// TIA Portal V16 export
// export: Created 2021-11-12T13:31:47.3064744Z, ExportSetting WithDefaults, DisplayName Totally Integrated Automation Portal, DisplayVersion V16 Update 3, DisplayName TIA Portal Version Control Interface, DisplayVersion V16 Update 2, DisplayName TIA Portal Openness, DisplayVersion V16 Update 3, DisplayName SINAMICS Startdrive Advanced, DisplayVersion V16 Update 5, DisplayName SINAMICS Startdrive G130, G150, S120, S150, SINAMICS MV, S210, DisplayVersion V16 Update 5, DisplayName SINAMICS Startdrive G110M, G120, G120C, G120D, G120P, G115D, DisplayVersion V16 Update 5, DisplayName STEP 7 Professional, DisplayVersion V16 Update 3, DisplayName STEP 7 Safety, DisplayVersion V16, DisplayName WinCC UA Professional, DisplayVersion V16 Update 3
FUNCTION_BLOCK "Zone000"   // FB72, LAD
{ S7_Optimized_Access := 'TRUE' }
VERSION : 0.1
// stored: AutoNumber true, IsIECCheckEnabled false, IsRetainMemResEnabled false, MemoryReserve 100, SetENOAutomatically false, UDAEnableTagReadback false
   VAR
      SF_StationMEM1Mode { S7_SetPoint := 'True'} : "STD_Station";
      "SF_EQ01-MA01" : "STD_Drive1";   // Čerpadlo cirkulace (P133) / Water pump (P51)
      "SF_EQ01-MA02" : "STD_Drive1";   // Čerpadlo cirkulace (P133) / Water pump (P52)
      "SF_EQ02-MA01" : "STD_Drive1";   // Čerpadlo cirkulace (P133) / Water pump (P61)
      "SF_UC11-TA01" { S7_SetPoint := 'True'} : "STD_Siemens_G120_CU240E_2_PN";   // Frekvenční měnič ( pro P33) / Frequence changer
      "SF_UC11-TA02" { S7_SetPoint := 'True'} : "STD_Siemens_G120_CU240E_2_PN";   // Frekvenční měnič ( pro P33) / Frequence changer
      "SF_UC11-TA03" { S7_SetPoint := 'True'} : "STD_Siemens_G120_CU240E_2_PN";   // Frekvenční měnič ( pro P33) / Frequence changer
      SS_Edge { S7_SetPoint := 'True'} : Array[0..100] of Bool;
      SB1_PowerOk { S7_SetPoint := 'True'} : Bool;
   END_VAR
   VAR_TEMP
      TS_EQ01MA01 : "UDT_DriveControl";   // Water pump (P51) / Čerpadlo cirkulace (P133)
      TS_EQ01MA02 : "UDT_DriveControl";   // Valve with servomotor (P52) / Ventil se servopohonem (A1419)
      TS_EQ02MA01 : "UDT_DriveControl";   // Valve with servomotor (P61) / Ventil se servopohonem (A1416)
      TS_UC11TA01 : Struct   // Frequence changer / Frekvenční měnič ( pro P33)
         ReqDir1 : Bool;   // Move in direction 1
         ReqDir2 : Bool;   // Move in direction 2
         AckErr : Bool;   // Acknowledge error
         SpeedSP : Real;   // Speed setpoint
      END_STRUCT;
      TS_UC11TA02 : Struct   // Frequence changer / Frekvenční měnič ( pro P33)
         ReqDir1 : Bool;   // Move in direction 1
         ReqDir2 : Bool;   // Move in direction 2
         AckErr : Bool;   // Acknowledge error
         SpeedSP : Real;   // Speed setpoint
      END_STRUCT;
      TS_UC11TA03 : Struct   // Frequence changer / Frekvenční měnič ( pro P33)
         ReqDir1 : Bool;   // Move in direction 1
         ReqDir2 : Bool;   // Move in direction 2
         AckErr : Bool;   // Acknowledge error
         SpeedSP : Real;   // Speed setpoint
      END_STRUCT;
   END_VAR
BEGIN

REGION Network 1: *************** Zone 000 ***************
END_REGION

REGION Network 2: Acknowledge from all zones
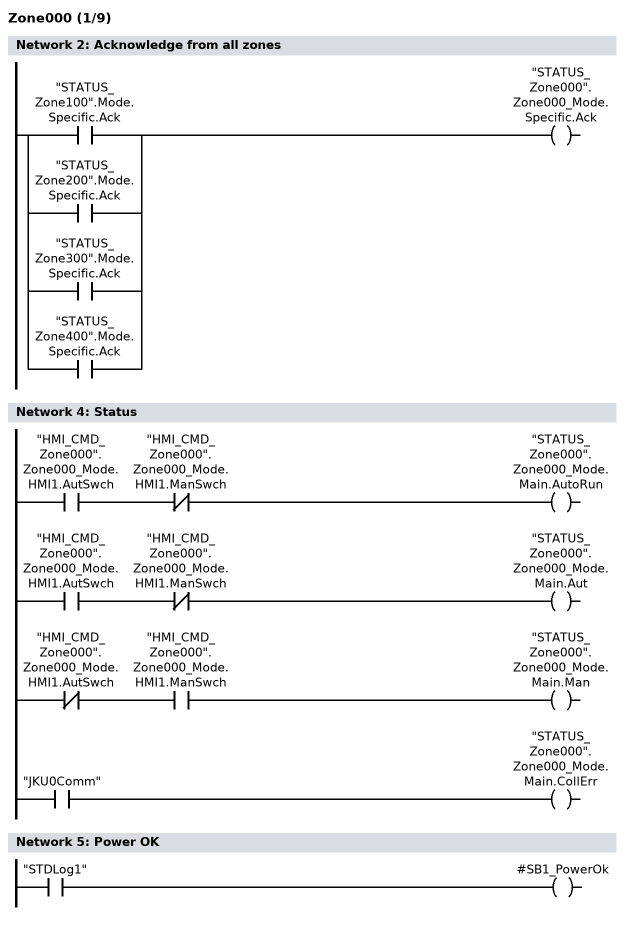
   RUNG wire#powerrail
      Contact( "STATUS_Zone100".Mode.Specific.Ack )
      wire#w1
      Coil( "STATUS_Zone000".Zone000_Mode.Specific.Ack )
   END_RUNG
   RUNG wire#powerrail
      Contact( "STATUS_Zone200".Mode.Specific.Ack )
   END_RUNG wire#w1
   RUNG wire#powerrail
      Contact( "STATUS_Zone300".Mode.Specific.Ack )
   END_RUNG wire#w1
   RUNG wire#powerrail
      Contact( "STATUS_Zone400".Mode.Specific.Ack )
   END_RUNG wire#w1
   // the same network as SCL:
   "STATUS_Zone000".Zone000_Mode.Specific.Ack := "STATUS_Zone100".Mode.Specific.Ack OR "STATUS_Zone200".Mode.Specific.Ack OR "STATUS_Zone300".Mode.Specific.Ack OR "STATUS_Zone400".Mode.Specific.Ack;
END_REGION

REGION Network 3: Alarms
END_REGION

REGION Network 4: Status
   RUNG wire#powerrail
      Contact( "HMI_CMD_Zone000".Zone000_Mode.HMI1.AutSwch )
      I_Contact( "HMI_CMD_Zone000".Zone000_Mode.HMI1.ManSwch )
      Coil( "STATUS_Zone000".Zone000_Mode.Main.AutoRun )
   END_RUNG
   RUNG wire#powerrail
      Contact( "HMI_CMD_Zone000".Zone000_Mode.HMI1.AutSwch )
      I_Contact( "HMI_CMD_Zone000".Zone000_Mode.HMI1.ManSwch )
      Coil( "STATUS_Zone000".Zone000_Mode.Main.Aut )
   END_RUNG
   RUNG wire#powerrail
      I_Contact( "HMI_CMD_Zone000".Zone000_Mode.HMI1.AutSwch )
      Contact( "HMI_CMD_Zone000".Zone000_Mode.HMI1.ManSwch )
      Coil( "STATUS_Zone000".Zone000_Mode.Main.Man )
   END_RUNG
   RUNG wire#powerrail
      Contact( "JKU0Comm" )
      Coil( "STATUS_Zone000".Zone000_Mode.Main.CollErr )
   END_RUNG
   // the same network as SCL:
   "STATUS_Zone000".Zone000_Mode.Main.AutoRun := "HMI_CMD_Zone000".Zone000_Mode.HMI1.AutSwch AND NOT "HMI_CMD_Zone000".Zone000_Mode.HMI1.ManSwch;
   "STATUS_Zone000".Zone000_Mode.Main.Aut := "HMI_CMD_Zone000".Zone000_Mode.HMI1.AutSwch AND NOT "HMI_CMD_Zone000".Zone000_Mode.HMI1.ManSwch;
   "STATUS_Zone000".Zone000_Mode.Main.Man := NOT "HMI_CMD_Zone000".Zone000_Mode.HMI1.AutSwch AND "HMI_CMD_Zone000".Zone000_Mode.HMI1.ManSwch;
   "STATUS_Zone000".Zone000_Mode.Main.CollErr := "JKU0Comm";
END_REGION

REGION Network 5: Power OK
   RUNG wire#powerrail
      Contact( "STDLog1" )
      Coil( #SB1_PowerOk )
   END_RUNG
   // the same network as SCL:
   #SB1_PowerOk := "STDLog1";
END_REGION

REGION Network 6: *************** MEM1 ***************
END_REGION

REGION Network 7: MEM1 - Main control
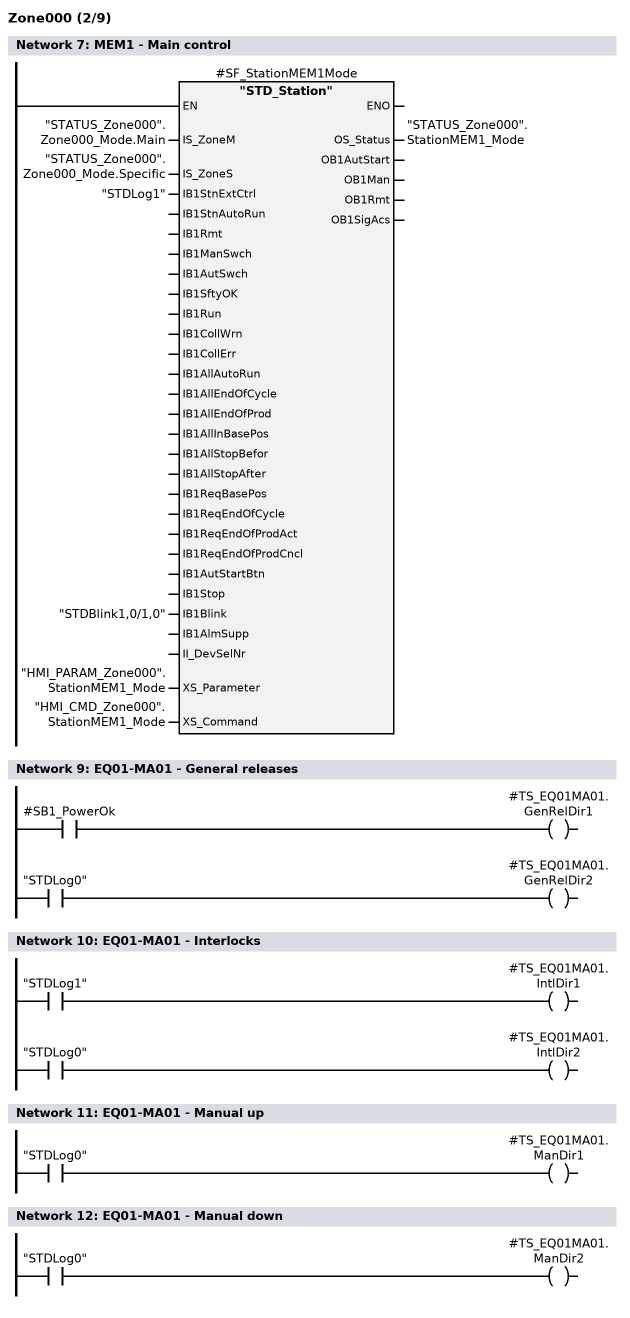
   RUNG wire#powerrail
      #SF_StationMEM1Mode(IS_ZoneM := "STATUS_Zone000".Zone000_Mode.Main, IS_ZoneS := "STATUS_Zone000".Zone000_Mode.Specific, IB1StnExtCtrl := "STDLog1", IB1StnAutoRun :=, IB1Rmt :=, IB1ManSwch :=, IB1AutSwch :=, IB1SftyOK :=, IB1Run :=, IB1CollWrn :=, IB1CollErr :=, IB1AllAutoRun :=, IB1AllEndOfCycle :=, IB1AllEndOfProd :=, IB1AllInBasePos :=, IB1AllStopBefor :=, IB1AllStopAfter :=, IB1ReqBasePos :=, IB1ReqEndOfCycle :=, IB1ReqEndOfProdAct :=, IB1ReqEndOfProdCncl :=, IB1AutStartBtn :=, IB1Stop :=, IB1Blink := "STDBlink1,0/1,0", IB1AlmSupp :=, II_DevSelNr :=, XS_Parameter := "HMI_PARAM_Zone000".StationMEM1_Mode, XS_Command := "HMI_CMD_Zone000".StationMEM1_Mode, OS_Status => "STATUS_Zone000".StationMEM1_Mode, OB1AutStart =>, OB1Man =>, OB1Rmt =>, OB1SigAcs =>)
   END_RUNG
   // the same network as SCL:
   #SF_StationMEM1Mode(IS_ZoneM := "STATUS_Zone000".Zone000_Mode.Main,   // "STD_Station"
                       IS_ZoneS := "STATUS_Zone000".Zone000_Mode.Specific,
                       IB1StnExtCtrl := "STDLog1",
                       IB1Blink := "STDBlink1,0/1,0",
                       XS_Parameter := "HMI_PARAM_Zone000".StationMEM1_Mode,
                       XS_Command := "HMI_CMD_Zone000".StationMEM1_Mode,
                       OS_Status => "STATUS_Zone000".StationMEM1_Mode);
END_REGION

REGION Network 8: ********** EQ01-MA01 **********
END_REGION

REGION Network 9: EQ01-MA01 - General releases
   RUNG wire#powerrail
      Contact( #SB1_PowerOk )
      Coil( #TS_EQ01MA01.GenRelDir1 )
   END_RUNG
   RUNG wire#powerrail
      Contact( "STDLog0" )
      Coil( #TS_EQ01MA01.GenRelDir2 )
   END_RUNG
   // the same network as SCL:
   #TS_EQ01MA01.GenRelDir1 := #SB1_PowerOk;
   #TS_EQ01MA01.GenRelDir2 := "STDLog0";
END_REGION

REGION Network 10: EQ01-MA01 - Interlocks
   RUNG wire#powerrail
      Contact( "STDLog1" )
      Coil( #TS_EQ01MA01.IntlDir1 )
   END_RUNG
   RUNG wire#powerrail
      Contact( "STDLog0" )
      Coil( #TS_EQ01MA01.IntlDir2 )
   END_RUNG
   // the same network as SCL:
   #TS_EQ01MA01.IntlDir1 := "STDLog1";
   #TS_EQ01MA01.IntlDir2 := "STDLog0";
END_REGION

REGION Network 11: EQ01-MA01 - Manual up
   RUNG wire#powerrail
      Contact( "STDLog0" )
      Coil( #TS_EQ01MA01.ManDir1 )
   END_RUNG
   // the same network as SCL:
   #TS_EQ01MA01.ManDir1 := "STDLog0";
END_REGION

REGION Network 12: EQ01-MA01 - Manual down
   RUNG wire#powerrail
      Contact( "STDLog0" )
      Coil( #TS_EQ01MA01.ManDir2 )
   END_RUNG
   // the same network as SCL:
   #TS_EQ01MA01.ManDir2 := "STDLog0";
END_REGION

REGION Network 13: EQ01-MA01 - Auto up
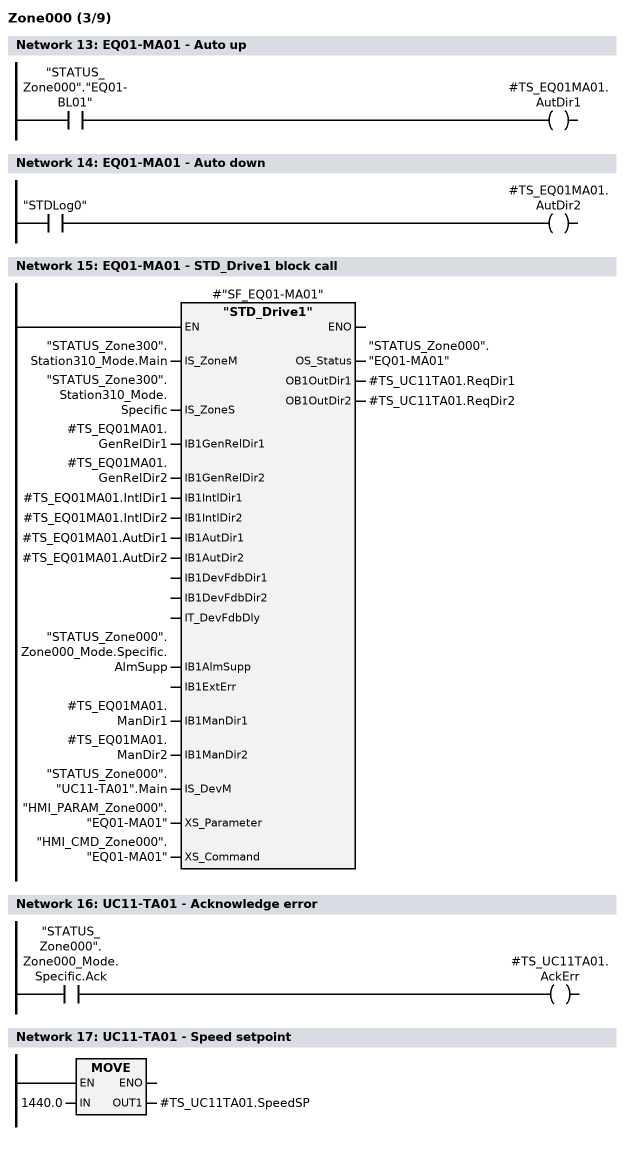
   RUNG wire#powerrail
      Contact( "STATUS_Zone000"."EQ01-BL01" )
      Coil( #TS_EQ01MA01.AutDir1 )
   END_RUNG
   // the same network as SCL:
   #TS_EQ01MA01.AutDir1 := "STATUS_Zone000"."EQ01-BL01";
END_REGION

REGION Network 14: EQ01-MA01 - Auto down
   RUNG wire#powerrail
      Contact( "STDLog0" )
      Coil( #TS_EQ01MA01.AutDir2 )
   END_RUNG
   // the same network as SCL:
   #TS_EQ01MA01.AutDir2 := "STDLog0";
END_REGION

REGION Network 15: EQ01-MA01 - STD_Drive1 block call
   RUNG wire#powerrail
      #"SF_EQ01-MA01"(IS_ZoneM := "STATUS_Zone300".Station310_Mode.Main, IS_ZoneS := "STATUS_Zone300".Station310_Mode.Specific, IB1GenRelDir1 := #TS_EQ01MA01.GenRelDir1, IB1GenRelDir2 := #TS_EQ01MA01.GenRelDir2, IB1IntlDir1 := #TS_EQ01MA01.IntlDir1, IB1IntlDir2 := #TS_EQ01MA01.IntlDir2, IB1AutDir1 := #TS_EQ01MA01.AutDir1, IB1AutDir2 := #TS_EQ01MA01.AutDir2, IB1DevFdbDir1 :=, IB1DevFdbDir2 :=, IT_DevFdbDly :=, IB1AlmSupp := "STATUS_Zone000".Zone000_Mode.Specific.AlmSupp, IB1ExtErr :=, IB1ManDir1 := #TS_EQ01MA01.ManDir1, IB1ManDir2 := #TS_EQ01MA01.ManDir2, IS_DevM := "STATUS_Zone000"."UC11-TA01".Main, XS_Parameter := "HMI_PARAM_Zone000"."EQ01-MA01", XS_Command := "HMI_CMD_Zone000"."EQ01-MA01", OS_Status => "STATUS_Zone000"."EQ01-MA01", OB1OutDir1 => #TS_UC11TA01.ReqDir1, OB1OutDir2 => #TS_UC11TA01.ReqDir2)
   END_RUNG
   // the same network as SCL:
   #"SF_EQ01-MA01"(IS_ZoneM := "STATUS_Zone300".Station310_Mode.Main,   // "STD_Drive1"
                   IS_ZoneS := "STATUS_Zone300".Station310_Mode.Specific,
                   IB1GenRelDir1 := #TS_EQ01MA01.GenRelDir1,
                   IB1GenRelDir2 := #TS_EQ01MA01.GenRelDir2,
                   IB1IntlDir1 := #TS_EQ01MA01.IntlDir1,
                   IB1IntlDir2 := #TS_EQ01MA01.IntlDir2,
                   IB1AutDir1 := #TS_EQ01MA01.AutDir1,
                   IB1AutDir2 := #TS_EQ01MA01.AutDir2,
                   IB1AlmSupp := "STATUS_Zone000".Zone000_Mode.Specific.AlmSupp,
                   IB1ManDir1 := #TS_EQ01MA01.ManDir1,
                   IB1ManDir2 := #TS_EQ01MA01.ManDir2,
                   IS_DevM := "STATUS_Zone000"."UC11-TA01".Main,
                   XS_Parameter := "HMI_PARAM_Zone000"."EQ01-MA01",
                   XS_Command := "HMI_CMD_Zone000"."EQ01-MA01",
                   OS_Status => "STATUS_Zone000"."EQ01-MA01",
                   OB1OutDir1 => #TS_UC11TA01.ReqDir1,
                   OB1OutDir2 => #TS_UC11TA01.ReqDir2);
END_REGION

REGION Network 16: UC11-TA01 - Acknowledge error
   RUNG wire#powerrail
      Contact( "STATUS_Zone000".Zone000_Mode.Specific.Ack )
      Coil( #TS_UC11TA01.AckErr )
   END_RUNG
   // the same network as SCL:
   #TS_UC11TA01.AckErr := "STATUS_Zone000".Zone000_Mode.Specific.Ack;
END_REGION

REGION Network 17: UC11-TA01 - Speed setpoint
   RUNG wire#powerrail
      Move(in := 1440.0, out1 => #TS_UC11TA01.SpeedSP)
   END_RUNG
   // the same network as SCL:
   #TS_UC11TA01.SpeedSP := 1440.0;
END_REGION

REGION Network 18: UC11-TA01 - Sinamics G120 STD block call (frequency convertor)
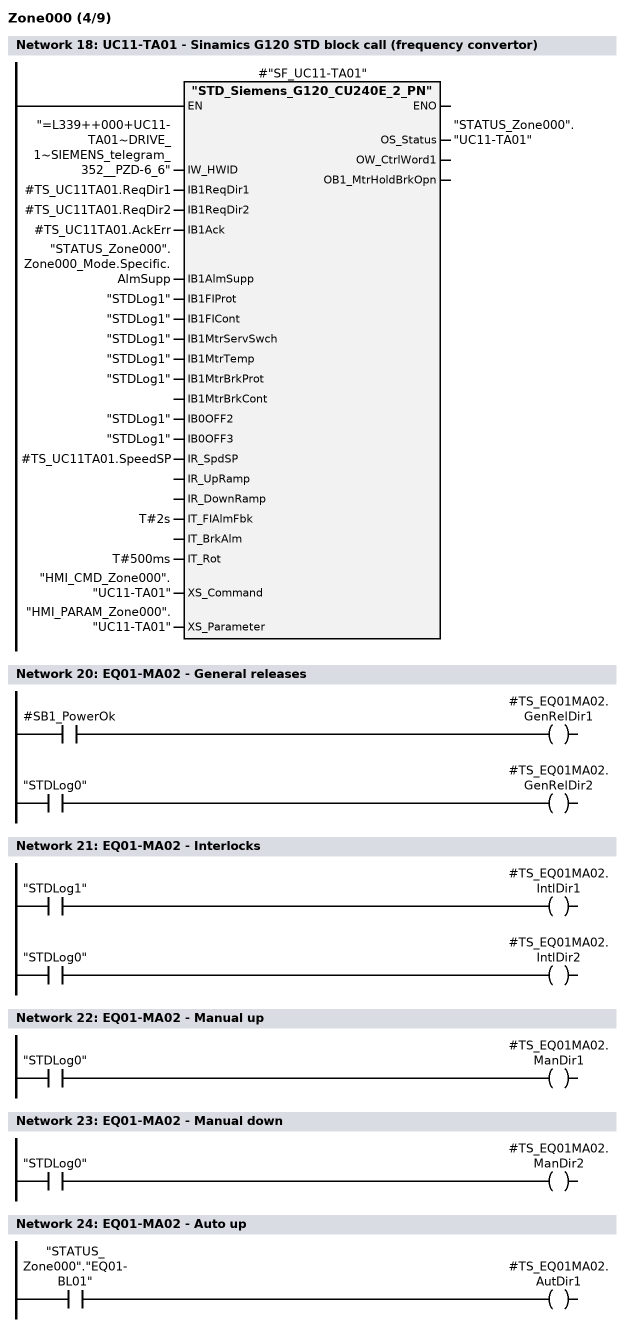
   RUNG wire#powerrail
      #"SF_UC11-TA01"(IW_HWID := "=L339++000+UC11-TA01~DRIVE_1~SIEMENS_telegram_352__PZD-6_6", IB1ReqDir1 := #TS_UC11TA01.ReqDir1, IB1ReqDir2 := #TS_UC11TA01.ReqDir2, IB1Ack := #TS_UC11TA01.AckErr, IB1AlmSupp := "STATUS_Zone000".Zone000_Mode.Specific.AlmSupp, IB1FIProt := "STDLog1", IB1FICont := "STDLog1", IB1MtrServSwch := "STDLog1", IB1MtrTemp := "STDLog1", IB1MtrBrkProt := "STDLog1", IB1MtrBrkCont :=, IB0OFF2 := "STDLog1", IB0OFF3 := "STDLog1", IR_SpdSP := #TS_UC11TA01.SpeedSP, IR_UpRamp :=, IR_DownRamp :=, IT_FIAlmFbk := T#2s, IT_BrkAlm :=, IT_Rot := T#500ms, XS_Command := "HMI_CMD_Zone000"."UC11-TA01", XS_Parameter := "HMI_PARAM_Zone000"."UC11-TA01", OS_Status => "STATUS_Zone000"."UC11-TA01", OW_CtrlWord1 =>, OB1_MtrHoldBrkOpn =>)
   END_RUNG
   // the same network as SCL:
   #"SF_UC11-TA01"(IW_HWID := "=L339++000+UC11-TA01~DRIVE_1~SIEMENS_telegram_352__PZD-6_6",   // "STD_Siemens_G120_CU240E_2_PN"
                   IB1ReqDir1 := #TS_UC11TA01.ReqDir1,
                   IB1ReqDir2 := #TS_UC11TA01.ReqDir2,
                   IB1Ack := #TS_UC11TA01.AckErr,
                   IB1AlmSupp := "STATUS_Zone000".Zone000_Mode.Specific.AlmSupp,
                   IB1FIProt := "STDLog1",
                   IB1FICont := "STDLog1",
                   IB1MtrServSwch := "STDLog1",
                   IB1MtrTemp := "STDLog1",
                   IB1MtrBrkProt := "STDLog1",
                   IB0OFF2 := "STDLog1",
                   IB0OFF3 := "STDLog1",
                   IR_SpdSP := #TS_UC11TA01.SpeedSP,
                   IT_FIAlmFbk := T#2s,
                   IT_Rot := T#500ms,
                   XS_Command := "HMI_CMD_Zone000"."UC11-TA01",
                   XS_Parameter := "HMI_PARAM_Zone000"."UC11-TA01",
                   OS_Status => "STATUS_Zone000"."UC11-TA01");
END_REGION

REGION Network 19: ********** EQ01-MA02 **********
END_REGION

REGION Network 20: EQ01-MA02 - General releases
   RUNG wire#powerrail
      Contact( #SB1_PowerOk )
      Coil( #TS_EQ01MA02.GenRelDir1 )
   END_RUNG
   RUNG wire#powerrail
      Contact( "STDLog0" )
      Coil( #TS_EQ01MA02.GenRelDir2 )
   END_RUNG
   // the same network as SCL:
   #TS_EQ01MA02.GenRelDir1 := #SB1_PowerOk;
   #TS_EQ01MA02.GenRelDir2 := "STDLog0";
END_REGION

REGION Network 21: EQ01-MA02 - Interlocks
   RUNG wire#powerrail
      Contact( "STDLog1" )
      Coil( #TS_EQ01MA02.IntlDir1 )
   END_RUNG
   RUNG wire#powerrail
      Contact( "STDLog0" )
      Coil( #TS_EQ01MA02.IntlDir2 )
   END_RUNG
   // the same network as SCL:
   #TS_EQ01MA02.IntlDir1 := "STDLog1";
   #TS_EQ01MA02.IntlDir2 := "STDLog0";
END_REGION

REGION Network 22: EQ01-MA02 - Manual up
   RUNG wire#powerrail
      Contact( "STDLog0" )
      Coil( #TS_EQ01MA02.ManDir1 )
   END_RUNG
   // the same network as SCL:
   #TS_EQ01MA02.ManDir1 := "STDLog0";
END_REGION

REGION Network 23: EQ01-MA02 - Manual down
   RUNG wire#powerrail
      Contact( "STDLog0" )
      Coil( #TS_EQ01MA02.ManDir2 )
   END_RUNG
   // the same network as SCL:
   #TS_EQ01MA02.ManDir2 := "STDLog0";
END_REGION

REGION Network 24: EQ01-MA02 - Auto up
   RUNG wire#powerrail
      Contact( "STATUS_Zone000"."EQ01-BL01" )
      Coil( #TS_EQ01MA02.AutDir1 )
   END_RUNG
   // the same network as SCL:
   #TS_EQ01MA02.AutDir1 := "STATUS_Zone000"."EQ01-BL01";
END_REGION

REGION Network 25: EQ01-MA02 - Auto down
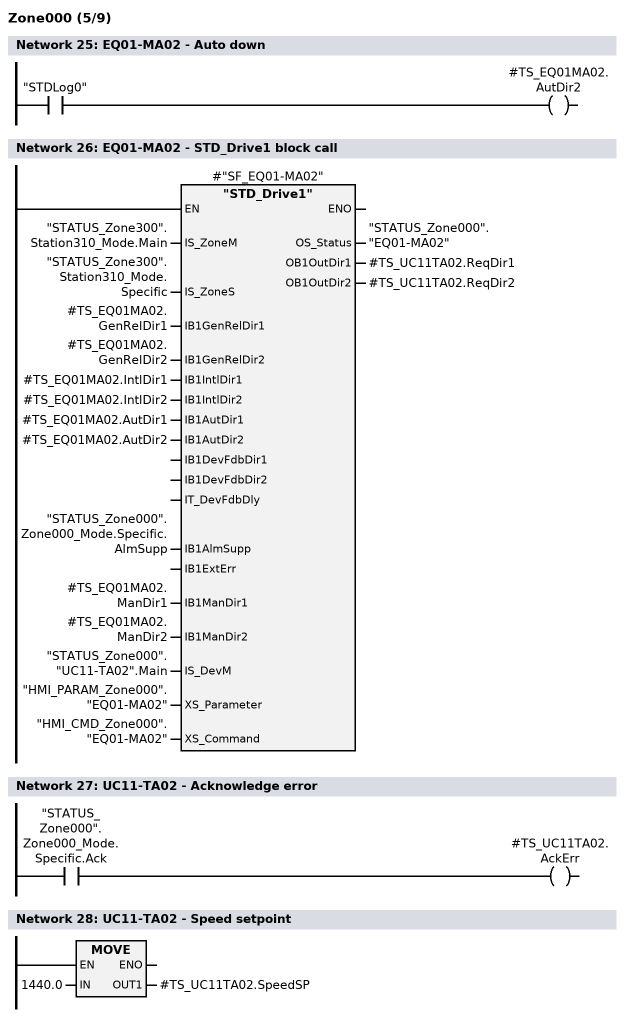
   RUNG wire#powerrail
      Contact( "STDLog0" )
      Coil( #TS_EQ01MA02.AutDir2 )
   END_RUNG
   // the same network as SCL:
   #TS_EQ01MA02.AutDir2 := "STDLog0";
END_REGION

REGION Network 26: EQ01-MA02 - STD_Drive1 block call
   RUNG wire#powerrail
      #"SF_EQ01-MA02"(IS_ZoneM := "STATUS_Zone300".Station310_Mode.Main, IS_ZoneS := "STATUS_Zone300".Station310_Mode.Specific, IB1GenRelDir1 := #TS_EQ01MA02.GenRelDir1, IB1GenRelDir2 := #TS_EQ01MA02.GenRelDir2, IB1IntlDir1 := #TS_EQ01MA02.IntlDir1, IB1IntlDir2 := #TS_EQ01MA02.IntlDir2, IB1AutDir1 := #TS_EQ01MA02.AutDir1, IB1AutDir2 := #TS_EQ01MA02.AutDir2, IB1DevFdbDir1 :=, IB1DevFdbDir2 :=, IT_DevFdbDly :=, IB1AlmSupp := "STATUS_Zone000".Zone000_Mode.Specific.AlmSupp, IB1ExtErr :=, IB1ManDir1 := #TS_EQ01MA02.ManDir1, IB1ManDir2 := #TS_EQ01MA02.ManDir2, IS_DevM := "STATUS_Zone000"."UC11-TA02".Main, XS_Parameter := "HMI_PARAM_Zone000"."EQ01-MA02", XS_Command := "HMI_CMD_Zone000"."EQ01-MA02", OS_Status => "STATUS_Zone000"."EQ01-MA02", OB1OutDir1 => #TS_UC11TA02.ReqDir1, OB1OutDir2 => #TS_UC11TA02.ReqDir2)
   END_RUNG
   // the same network as SCL:
   #"SF_EQ01-MA02"(IS_ZoneM := "STATUS_Zone300".Station310_Mode.Main,   // "STD_Drive1"
                   IS_ZoneS := "STATUS_Zone300".Station310_Mode.Specific,
                   IB1GenRelDir1 := #TS_EQ01MA02.GenRelDir1,
                   IB1GenRelDir2 := #TS_EQ01MA02.GenRelDir2,
                   IB1IntlDir1 := #TS_EQ01MA02.IntlDir1,
                   IB1IntlDir2 := #TS_EQ01MA02.IntlDir2,
                   IB1AutDir1 := #TS_EQ01MA02.AutDir1,
                   IB1AutDir2 := #TS_EQ01MA02.AutDir2,
                   IB1AlmSupp := "STATUS_Zone000".Zone000_Mode.Specific.AlmSupp,
                   IB1ManDir1 := #TS_EQ01MA02.ManDir1,
                   IB1ManDir2 := #TS_EQ01MA02.ManDir2,
                   IS_DevM := "STATUS_Zone000"."UC11-TA02".Main,
                   XS_Parameter := "HMI_PARAM_Zone000"."EQ01-MA02",
                   XS_Command := "HMI_CMD_Zone000"."EQ01-MA02",
                   OS_Status => "STATUS_Zone000"."EQ01-MA02",
                   OB1OutDir1 => #TS_UC11TA02.ReqDir1,
                   OB1OutDir2 => #TS_UC11TA02.ReqDir2);
END_REGION

REGION Network 27: UC11-TA02 - Acknowledge error
   RUNG wire#powerrail
      Contact( "STATUS_Zone000".Zone000_Mode.Specific.Ack )
      Coil( #TS_UC11TA02.AckErr )
   END_RUNG
   // the same network as SCL:
   #TS_UC11TA02.AckErr := "STATUS_Zone000".Zone000_Mode.Specific.Ack;
END_REGION

REGION Network 28: UC11-TA02 - Speed setpoint
   RUNG wire#powerrail
      Move(in := 1440.0, out1 => #TS_UC11TA02.SpeedSP)
   END_RUNG
   // the same network as SCL:
   #TS_UC11TA02.SpeedSP := 1440.0;
END_REGION

REGION Network 29: UC11-TA02 - Sinamics G120 STD block call (frequency convertor)
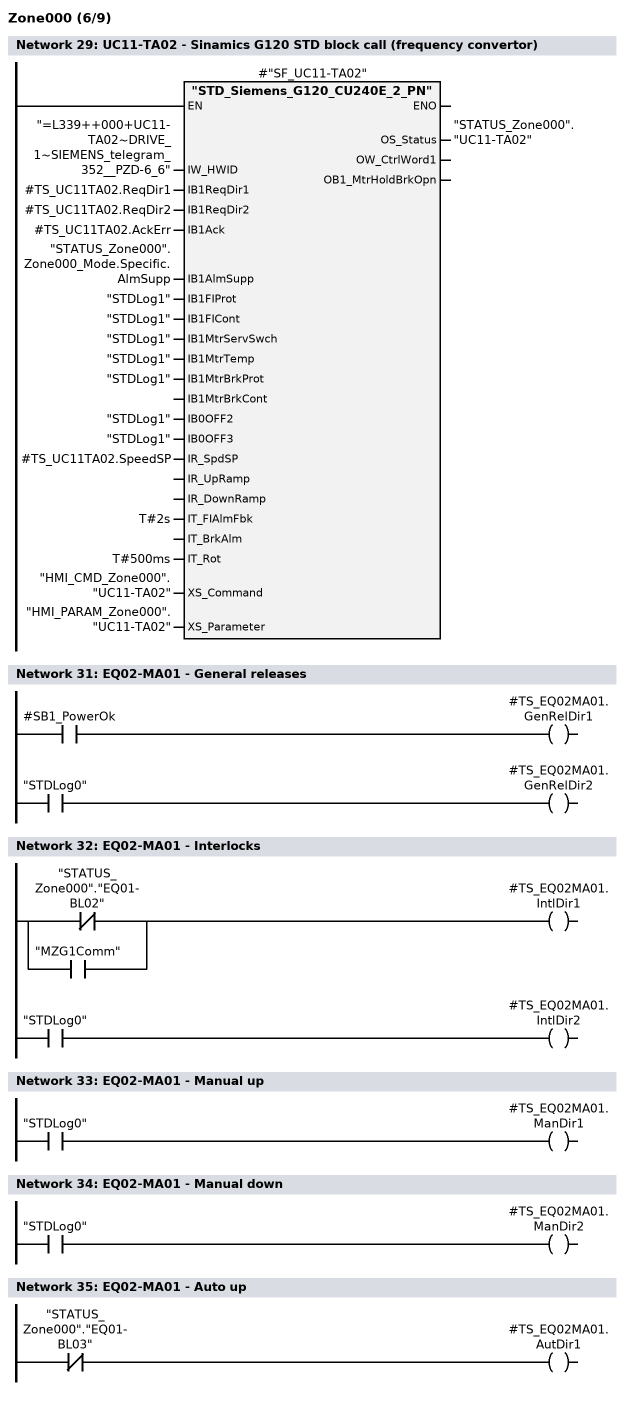
   RUNG wire#powerrail
      #"SF_UC11-TA02"(IW_HWID := "=L339++000+UC11-TA02~DRIVE_1~SIEMENS_telegram_352__PZD-6_6", IB1ReqDir1 := #TS_UC11TA02.ReqDir1, IB1ReqDir2 := #TS_UC11TA02.ReqDir2, IB1Ack := #TS_UC11TA02.AckErr, IB1AlmSupp := "STATUS_Zone000".Zone000_Mode.Specific.AlmSupp, IB1FIProt := "STDLog1", IB1FICont := "STDLog1", IB1MtrServSwch := "STDLog1", IB1MtrTemp := "STDLog1", IB1MtrBrkProt := "STDLog1", IB1MtrBrkCont :=, IB0OFF2 := "STDLog1", IB0OFF3 := "STDLog1", IR_SpdSP := #TS_UC11TA02.SpeedSP, IR_UpRamp :=, IR_DownRamp :=, IT_FIAlmFbk := T#2s, IT_BrkAlm :=, IT_Rot := T#500ms, XS_Command := "HMI_CMD_Zone000"."UC11-TA02", XS_Parameter := "HMI_PARAM_Zone000"."UC11-TA02", OS_Status => "STATUS_Zone000"."UC11-TA02", OW_CtrlWord1 =>, OB1_MtrHoldBrkOpn =>)
   END_RUNG
   // the same network as SCL:
   #"SF_UC11-TA02"(IW_HWID := "=L339++000+UC11-TA02~DRIVE_1~SIEMENS_telegram_352__PZD-6_6",   // "STD_Siemens_G120_CU240E_2_PN"
                   IB1ReqDir1 := #TS_UC11TA02.ReqDir1,
                   IB1ReqDir2 := #TS_UC11TA02.ReqDir2,
                   IB1Ack := #TS_UC11TA02.AckErr,
                   IB1AlmSupp := "STATUS_Zone000".Zone000_Mode.Specific.AlmSupp,
                   IB1FIProt := "STDLog1",
                   IB1FICont := "STDLog1",
                   IB1MtrServSwch := "STDLog1",
                   IB1MtrTemp := "STDLog1",
                   IB1MtrBrkProt := "STDLog1",
                   IB0OFF2 := "STDLog1",
                   IB0OFF3 := "STDLog1",
                   IR_SpdSP := #TS_UC11TA02.SpeedSP,
                   IT_FIAlmFbk := T#2s,
                   IT_Rot := T#500ms,
                   XS_Command := "HMI_CMD_Zone000"."UC11-TA02",
                   XS_Parameter := "HMI_PARAM_Zone000"."UC11-TA02",
                   OS_Status => "STATUS_Zone000"."UC11-TA02");
END_REGION

REGION Network 30: ********** EQ02-MA01 **********
END_REGION

REGION Network 31: EQ02-MA01 - General releases
   RUNG wire#powerrail
      Contact( #SB1_PowerOk )
      Coil( #TS_EQ02MA01.GenRelDir1 )
   END_RUNG
   RUNG wire#powerrail
      Contact( "STDLog0" )
      Coil( #TS_EQ02MA01.GenRelDir2 )
   END_RUNG
   // the same network as SCL:
   #TS_EQ02MA01.GenRelDir1 := #SB1_PowerOk;
   #TS_EQ02MA01.GenRelDir2 := "STDLog0";
END_REGION

REGION Network 32: EQ02-MA01 - Interlocks
   RUNG wire#powerrail
      I_Contact( "STATUS_Zone000"."EQ01-BL02" )
      wire#w1
      Coil( #TS_EQ02MA01.IntlDir1 )
   END_RUNG
   RUNG wire#powerrail
      Contact( "MZG1Comm" )
   END_RUNG wire#w1
   RUNG wire#powerrail
      Contact( "STDLog0" )
      Coil( #TS_EQ02MA01.IntlDir2 )
   END_RUNG
   // the same network as SCL:
   #TS_EQ02MA01.IntlDir1 := NOT "STATUS_Zone000"."EQ01-BL02" OR "MZG1Comm";
   #TS_EQ02MA01.IntlDir2 := "STDLog0";
END_REGION

REGION Network 33: EQ02-MA01 - Manual up
   RUNG wire#powerrail
      Contact( "STDLog0" )
      Coil( #TS_EQ02MA01.ManDir1 )
   END_RUNG
   // the same network as SCL:
   #TS_EQ02MA01.ManDir1 := "STDLog0";
END_REGION

REGION Network 34: EQ02-MA01 - Manual down
   RUNG wire#powerrail
      Contact( "STDLog0" )
      Coil( #TS_EQ02MA01.ManDir2 )
   END_RUNG
   // the same network as SCL:
   #TS_EQ02MA01.ManDir2 := "STDLog0";
END_REGION

REGION Network 35: EQ02-MA01 - Auto up
   RUNG wire#powerrail
      I_Contact( "STATUS_Zone000"."EQ01-BL03" )
      Coil( #TS_EQ02MA01.AutDir1 )
   END_RUNG
   // the same network as SCL:
   #TS_EQ02MA01.AutDir1 := NOT "STATUS_Zone000"."EQ01-BL03";
END_REGION

REGION Network 36: EQ02-MA01 - Auto down
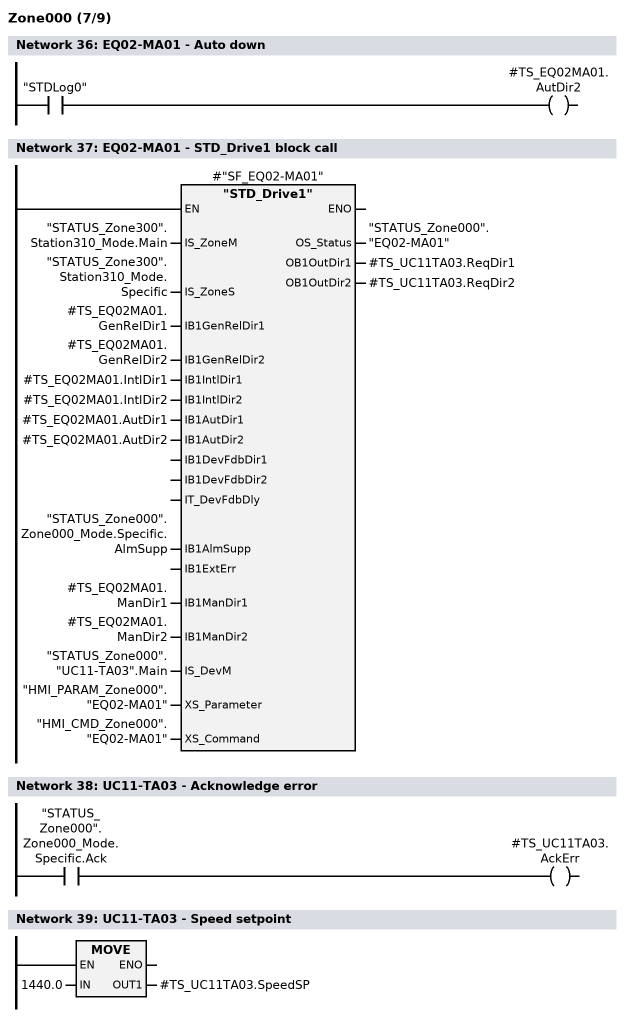
   RUNG wire#powerrail
      Contact( "STDLog0" )
      Coil( #TS_EQ02MA01.AutDir2 )
   END_RUNG
   // the same network as SCL:
   #TS_EQ02MA01.AutDir2 := "STDLog0";
END_REGION

REGION Network 37: EQ02-MA01 - STD_Drive1 block call
   RUNG wire#powerrail
      #"SF_EQ02-MA01"(IS_ZoneM := "STATUS_Zone300".Station310_Mode.Main, IS_ZoneS := "STATUS_Zone300".Station310_Mode.Specific, IB1GenRelDir1 := #TS_EQ02MA01.GenRelDir1, IB1GenRelDir2 := #TS_EQ02MA01.GenRelDir2, IB1IntlDir1 := #TS_EQ02MA01.IntlDir1, IB1IntlDir2 := #TS_EQ02MA01.IntlDir2, IB1AutDir1 := #TS_EQ02MA01.AutDir1, IB1AutDir2 := #TS_EQ02MA01.AutDir2, IB1DevFdbDir1 :=, IB1DevFdbDir2 :=, IT_DevFdbDly :=, IB1AlmSupp := "STATUS_Zone000".Zone000_Mode.Specific.AlmSupp, IB1ExtErr :=, IB1ManDir1 := #TS_EQ02MA01.ManDir1, IB1ManDir2 := #TS_EQ02MA01.ManDir2, IS_DevM := "STATUS_Zone000"."UC11-TA03".Main, XS_Parameter := "HMI_PARAM_Zone000"."EQ02-MA01", XS_Command := "HMI_CMD_Zone000"."EQ02-MA01", OS_Status => "STATUS_Zone000"."EQ02-MA01", OB1OutDir1 => #TS_UC11TA03.ReqDir1, OB1OutDir2 => #TS_UC11TA03.ReqDir2)
   END_RUNG
   // the same network as SCL:
   #"SF_EQ02-MA01"(IS_ZoneM := "STATUS_Zone300".Station310_Mode.Main,   // "STD_Drive1"
                   IS_ZoneS := "STATUS_Zone300".Station310_Mode.Specific,
                   IB1GenRelDir1 := #TS_EQ02MA01.GenRelDir1,
                   IB1GenRelDir2 := #TS_EQ02MA01.GenRelDir2,
                   IB1IntlDir1 := #TS_EQ02MA01.IntlDir1,
                   IB1IntlDir2 := #TS_EQ02MA01.IntlDir2,
                   IB1AutDir1 := #TS_EQ02MA01.AutDir1,
                   IB1AutDir2 := #TS_EQ02MA01.AutDir2,
                   IB1AlmSupp := "STATUS_Zone000".Zone000_Mode.Specific.AlmSupp,
                   IB1ManDir1 := #TS_EQ02MA01.ManDir1,
                   IB1ManDir2 := #TS_EQ02MA01.ManDir2,
                   IS_DevM := "STATUS_Zone000"."UC11-TA03".Main,
                   XS_Parameter := "HMI_PARAM_Zone000"."EQ02-MA01",
                   XS_Command := "HMI_CMD_Zone000"."EQ02-MA01",
                   OS_Status => "STATUS_Zone000"."EQ02-MA01",
                   OB1OutDir1 => #TS_UC11TA03.ReqDir1,
                   OB1OutDir2 => #TS_UC11TA03.ReqDir2);
END_REGION

REGION Network 38: UC11-TA03 - Acknowledge error
   RUNG wire#powerrail
      Contact( "STATUS_Zone000".Zone000_Mode.Specific.Ack )
      Coil( #TS_UC11TA03.AckErr )
   END_RUNG
   // the same network as SCL:
   #TS_UC11TA03.AckErr := "STATUS_Zone000".Zone000_Mode.Specific.Ack;
END_REGION

REGION Network 39: UC11-TA03 - Speed setpoint
   RUNG wire#powerrail
      Move(in := 1440.0, out1 => #TS_UC11TA03.SpeedSP)
   END_RUNG
   // the same network as SCL:
   #TS_UC11TA03.SpeedSP := 1440.0;
END_REGION

REGION Network 40: UC11-TA03 - Sinamics G120 STD block call (frequency convertor)
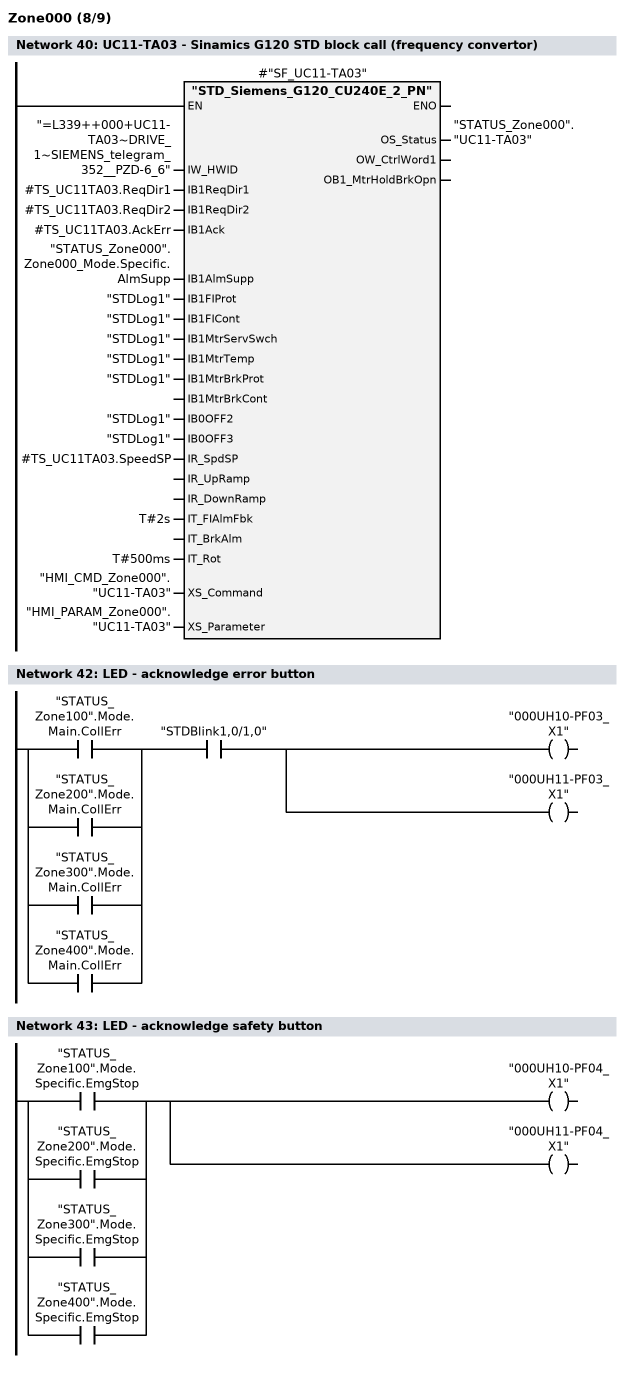
   RUNG wire#powerrail
      #"SF_UC11-TA03"(IW_HWID := "=L339++000+UC11-TA03~DRIVE_1~SIEMENS_telegram_352__PZD-6_6", IB1ReqDir1 := #TS_UC11TA03.ReqDir1, IB1ReqDir2 := #TS_UC11TA03.ReqDir2, IB1Ack := #TS_UC11TA03.AckErr, IB1AlmSupp := "STATUS_Zone000".Zone000_Mode.Specific.AlmSupp, IB1FIProt := "STDLog1", IB1FICont := "STDLog1", IB1MtrServSwch := "STDLog1", IB1MtrTemp := "STDLog1", IB1MtrBrkProt := "STDLog1", IB1MtrBrkCont :=, IB0OFF2 := "STDLog1", IB0OFF3 := "STDLog1", IR_SpdSP := #TS_UC11TA03.SpeedSP, IR_UpRamp :=, IR_DownRamp :=, IT_FIAlmFbk := T#2s, IT_BrkAlm :=, IT_Rot := T#500ms, XS_Command := "HMI_CMD_Zone000"."UC11-TA03", XS_Parameter := "HMI_PARAM_Zone000"."UC11-TA03", OS_Status => "STATUS_Zone000"."UC11-TA03", OW_CtrlWord1 =>, OB1_MtrHoldBrkOpn =>)
   END_RUNG
   // the same network as SCL:
   #"SF_UC11-TA03"(IW_HWID := "=L339++000+UC11-TA03~DRIVE_1~SIEMENS_telegram_352__PZD-6_6",   // "STD_Siemens_G120_CU240E_2_PN"
                   IB1ReqDir1 := #TS_UC11TA03.ReqDir1,
                   IB1ReqDir2 := #TS_UC11TA03.ReqDir2,
                   IB1Ack := #TS_UC11TA03.AckErr,
                   IB1AlmSupp := "STATUS_Zone000".Zone000_Mode.Specific.AlmSupp,
                   IB1FIProt := "STDLog1",
                   IB1FICont := "STDLog1",
                   IB1MtrServSwch := "STDLog1",
                   IB1MtrTemp := "STDLog1",
                   IB1MtrBrkProt := "STDLog1",
                   IB0OFF2 := "STDLog1",
                   IB0OFF3 := "STDLog1",
                   IR_SpdSP := #TS_UC11TA03.SpeedSP,
                   IT_FIAlmFbk := T#2s,
                   IT_Rot := T#500ms,
                   XS_Command := "HMI_CMD_Zone000"."UC11-TA03",
                   XS_Parameter := "HMI_PARAM_Zone000"."UC11-TA03",
                   OS_Status => "STATUS_Zone000"."UC11-TA03");
END_REGION

REGION Network 41: *************** Central panel button LEDs ***************
END_REGION

REGION Network 42: LED - acknowledge error button
   RUNG wire#powerrail
      Contact( "STATUS_Zone100".Mode.Main.CollErr )
      wire#w1
      Contact( "STDBlink1,0/1,0" )
      wire#w2
      Coil( "000UH10-PF03_X1" )
   END_RUNG
   RUNG wire#powerrail
      Contact( "STATUS_Zone200".Mode.Main.CollErr )
   END_RUNG wire#w1
   RUNG wire#powerrail
      Contact( "STATUS_Zone300".Mode.Main.CollErr )
   END_RUNG wire#w1
   RUNG wire#powerrail
      Contact( "STATUS_Zone400".Mode.Main.CollErr )
   END_RUNG wire#w1
   RUNG wire#w2
      Coil( "000UH11-PF03_X1" )
   END_RUNG
   // the same network as SCL:
   "000UH10-PF03_X1" := ("STATUS_Zone100".Mode.Main.CollErr OR "STATUS_Zone200".Mode.Main.CollErr OR "STATUS_Zone300".Mode.Main.CollErr OR "STATUS_Zone400".Mode.Main.CollErr) AND "STDBlink1,0/1,0";
   "000UH11-PF03_X1" := "000UH10-PF03_X1";
END_REGION

REGION Network 43: LED - acknowledge safety button
   RUNG wire#powerrail
      Contact( "STATUS_Zone100".Mode.Specific.EmgStop )
      wire#w1
      Coil( "000UH10-PF04_X1" )
   END_RUNG
   RUNG wire#powerrail
      Contact( "STATUS_Zone200".Mode.Specific.EmgStop )
   END_RUNG wire#w1
   RUNG wire#powerrail
      Contact( "STATUS_Zone300".Mode.Specific.EmgStop )
   END_RUNG wire#w1
   RUNG wire#powerrail
      Contact( "STATUS_Zone400".Mode.Specific.EmgStop )
   END_RUNG wire#w1
   RUNG wire#w1
      Coil( "000UH11-PF04_X1" )
   END_RUNG
   // the same network as SCL:
   "000UH10-PF04_X1" := "STATUS_Zone100".Mode.Specific.EmgStop OR "STATUS_Zone200".Mode.Specific.EmgStop OR "STATUS_Zone300".Mode.Specific.EmgStop OR "STATUS_Zone400".Mode.Specific.EmgStop;
   "000UH11-PF04_X1" := "000UH10-PF04_X1";
END_REGION

REGION Network 44: LED - automat start button
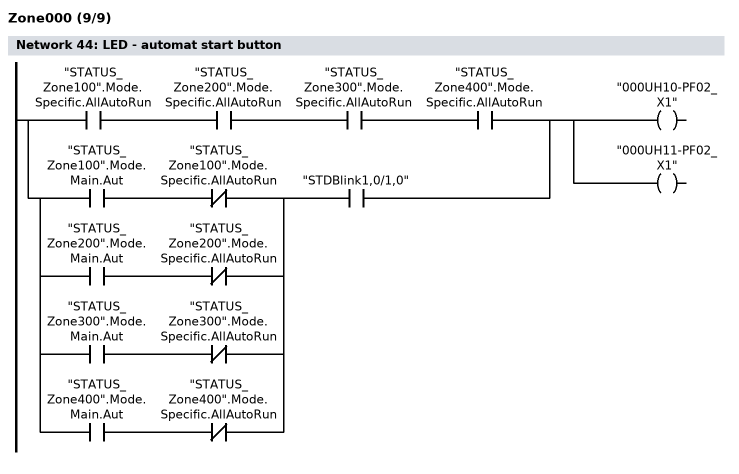
   RUNG wire#powerrail
      Contact( "STATUS_Zone100".Mode.Specific.AllAutoRun )
      Contact( "STATUS_Zone200".Mode.Specific.AllAutoRun )
      Contact( "STATUS_Zone300".Mode.Specific.AllAutoRun )
      Contact( "STATUS_Zone400".Mode.Specific.AllAutoRun )
      wire#w1
      Coil( "000UH10-PF02_X1" )
   END_RUNG
   RUNG wire#powerrail
      Contact( "STATUS_Zone100".Mode.Main.Aut )
      I_Contact( "STATUS_Zone100".Mode.Specific.AllAutoRun )
      wire#w2
      Contact( "STDBlink1,0/1,0" )
   END_RUNG wire#w1
   RUNG wire#powerrail
      Contact( "STATUS_Zone200".Mode.Main.Aut )
      I_Contact( "STATUS_Zone200".Mode.Specific.AllAutoRun )
   END_RUNG wire#w2
   RUNG wire#powerrail
      Contact( "STATUS_Zone300".Mode.Main.Aut )
      I_Contact( "STATUS_Zone300".Mode.Specific.AllAutoRun )
   END_RUNG wire#w2
   RUNG wire#powerrail
      Contact( "STATUS_Zone400".Mode.Main.Aut )
      I_Contact( "STATUS_Zone400".Mode.Specific.AllAutoRun )
   END_RUNG wire#w2
   RUNG wire#w1
      Coil( "000UH11-PF02_X1" )
   END_RUNG
   // the same network as SCL:
   "000UH10-PF02_X1" := ("STATUS_Zone100".Mode.Specific.AllAutoRun AND "STATUS_Zone200".Mode.Specific.AllAutoRun AND "STATUS_Zone300".Mode.Specific.AllAutoRun AND "STATUS_Zone400".Mode.Specific.AllAutoRun) OR ((("STATUS_Zone100".Mode.Main.Aut AND NOT "STATUS_Zone100".Mode.Specific.AllAutoRun) OR ("STATUS_Zone200".Mode.Main.Aut AND NOT "STATUS_Zone200".Mode.Specific.AllAutoRun) OR ("STATUS_Zone300".Mode.Main.Aut AND NOT "STATUS_Zone300".Mode.Specific.AllAutoRun) OR ("STATUS_Zone400".Mode.Main.Aut AND NOT "STATUS_Zone400".Mode.Specific.AllAutoRun)) AND "STDBlink1,0/1,0");
   "000UH11-PF02_X1" := "000UH10-PF02_X1";
END_REGION
END_FUNCTION_BLOCK
